TYPE DUT_SENSOR_DATAS_1 :
UNION
	data_lreal:REAL;
	data_byte:ARRAY[0..3] OF BYTE;
END_UNION
END_TYPE

(* stored: Version 1.1.0.1, ProductVersion 3.1.4024.6
   DUT DUT_SENSOR_DATAS_1: Id {53e42742-5f31-495f-b27b-a97d393542f2} *)
